// TIA Portal V14 SP1 export
// export: Created 2019-08-12T05:39:51.1994735Z, ExportSetting WithDefaults, WithReadOnly, DisplayName Totally Integrated Automation Portal, DisplayVersion V14 SP1 Update 6, DisplayName TIA Portal Openness, DisplayVersion V14 SP1 Update 6, DisplayName STEP 7 Professional, DisplayVersion V14 SP1 Update 6, DisplayName WinCC Professional, DisplayVersion V14 SP1 Update 6
FUNCTION_BLOCK "181M_Vibrating_screen"   // FB2008, LAD
TITLE = Управление виброситом силосов муки
{ S7_Optimized_Access := 'FALSE' }
VERSION : 0.1
// stored: AutoNumber false, CodeModifiedDate 2019-08-12T05:39:33.4572424Z, CompileDate 2019-08-12T05:39:33.4572423Z, CreationDate 2019-02-26T05:18:41.6523018Z, InterfaceModifiedDate 2019-08-09T12:59:29.73599Z, IsConsistent true, IsIECCheckEnabled false, IsKnowHowProtected false, ISMultiInstanceCapable true, IsWriteProtected false, LibraryConformanceStatus Warning: The object contains access to global data blocks. Warning: The block contains direct access to inputs, outputs, bit memories, indirect access to the registry or indirect access to external memory areas that are unknown at the time of compilation., ModifiedDate 2019-08-12T05:39:33.4572424Z, ParameterModified 2018-04-23T08:12:13.0838357Z, StructureModified 2019-08-09T12:59:29.73599Z, UDAEnableTagReadback false
   VAR DB_SPECIFIC
      HMI : Struct
         CMD : Struct
            Rot_FWD : Bool;   // Команда Вращение вперёд
            Stop : Bool;   // Команда Стоп
            Rot_BWD : Bool;   // Команда Вращение назад
            Spare_3 : Bool;
            Spare_4 : Bool;
            Spare_5 : Bool;
            Manual : Bool;   // Ручной режим
            Reset_Error : Bool;   // Сброс ошибок
         END_STRUCT;
         DATA : Struct
            StatusWord : Word;
            ContFbk1_Time : DInt := 4;   // Время контроля срабатывания контактора 1 / Время контроля срабатывания контактора 1 (сек)
            ContFbk2_Time : DInt := 4;   // Время контроля срабатывания контактора 2 / Время контроля срабатывания контактора 2 (сек)
            Rot_Off_Time : Int;   // Обратный отсчет времени остановки
            Warn_Not_Open_Valve : Bool;   // Сообщение о запуске очистки при закрытом клапане
            Warn_Not_Close_Valve : Bool;   // Сообщение о запуске работы при открытом клапане
         END_STRUCT;
      END_STRUCT;
   END_VAR
   VAR
      Two_Motor : "TwoMotorManag";
      TOF_Rot_FWD : TOF;
      TOF_Rot_REV : TOF;
   END_VAR
   VAR DB_SPECIFIC
      ContFbk1_Time : Time;   // Время контроля срабатывания контактора 1
      ContFbk2_Time : Time;   // Время контроля срабатывания контактора 2
      StopTime : Time;   // Время остановки мотора после вращения
      ResetErr : Bool;   // сброс ошибок
      General_cond_OK : Bool;   // Разрешение работы
      ManCmd_FWD : Bool;   // Команда ручного включения вращение вперёд
      ManCmd_REV : Bool;   // Команда ручного включения вращение назад
      ManCmd_Stop : Bool;   // Стоп
      AutoCmd_FWD : Bool;   // Команда автом. включения вращение вперёд
      AutoCmd_REV : Bool;   // Команда автом. включения вращение назад
      Spare : Bool;
      Spare_1 : Bool;
      Spare_2 : Bool;
      Spare_3 : Bool;
      Spare_4 : Bool;
      Spare_5 : Bool;
   END_VAR
   VAR_TEMP
      Temp_DINT : DInt;
   END_VAR
   VAR_TEMP   // added for the SCL form of the ladder/FBD networks
      _w1 : Bool;
   END_VAR
BEGIN

REGION Network 1: Сброс ошибок
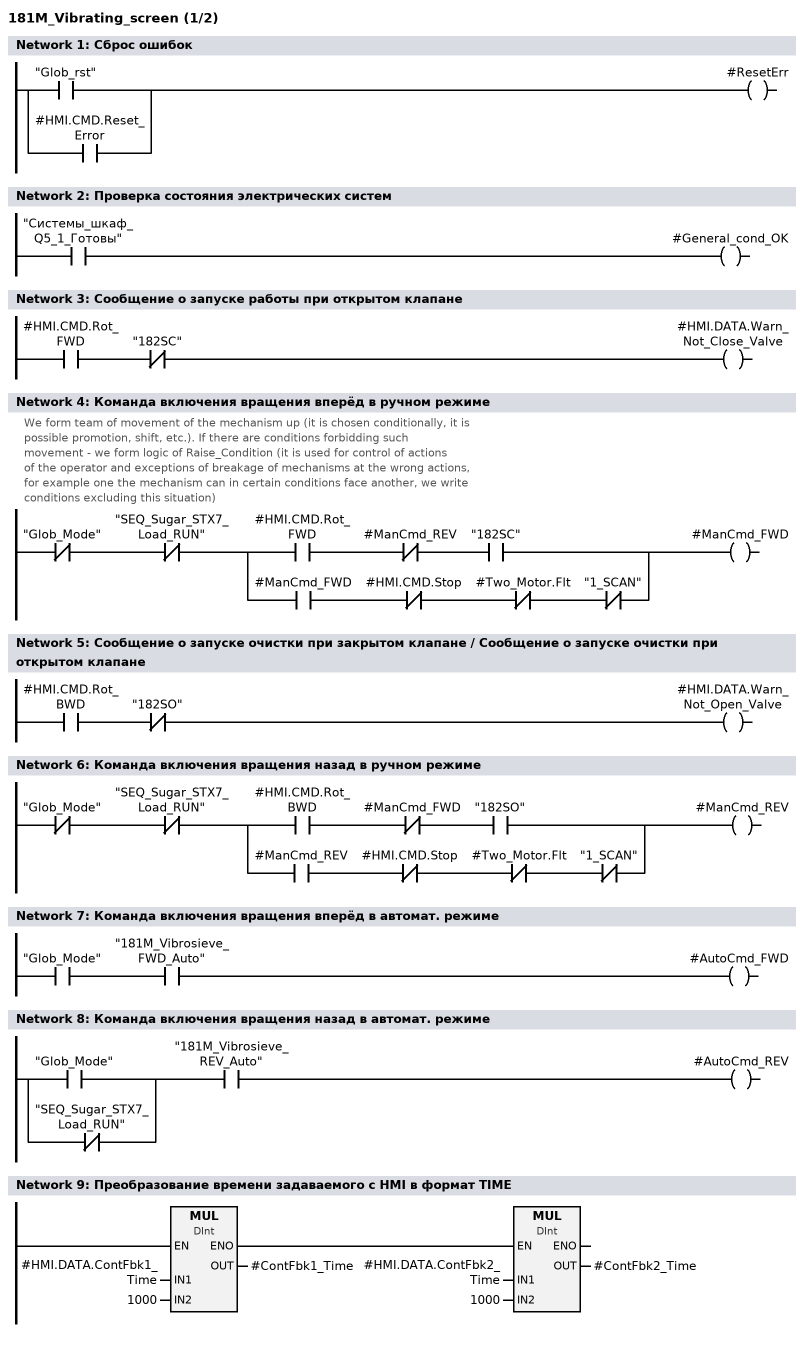
   RUNG wire#powerrail
      Contact( "Glob_rst" )
      wire#w1
      Coil( #ResetErr )
   END_RUNG
   RUNG wire#powerrail
      Contact( #HMI.CMD.Reset_Error )
   END_RUNG wire#w1
   // the same network as SCL:
   #ResetErr := "Glob_rst" OR #HMI.CMD.Reset_Error;
END_REGION

REGION Network 2: Проверка состояния электрических систем
   RUNG wire#powerrail
      Contact( "Системы_шкаф_Q5_1_Готовы" )
      Coil( #General_cond_OK )
   END_RUNG
   // the same network as SCL:
   #General_cond_OK := "Системы_шкаф_Q5_1_Готовы";
END_REGION

REGION Network 3: Сообщение о запуске работы при открытом клапане
   RUNG wire#powerrail
      Contact( #HMI.CMD.Rot_FWD )
      I_Contact( "182SC" )
      Coil( #HMI.DATA.Warn_Not_Close_Valve )
   END_RUNG
   // the same network as SCL:
   #HMI.DATA.Warn_Not_Close_Valve := #HMI.CMD.Rot_FWD AND NOT "182SC";
END_REGION

REGION Network 4: Команда включения вращения вперёд в ручном режиме
   // We form team of movement of the mechanism up (it is chosen conditionally, it is 
   // possible promotion, shift, etc.). If there are conditions forbidding such 
   // movement - we form logic of Raise_Condition (it is used for control of actions 
   // of the operator and exceptions of breakage of mechanisms at the wrong actions, 
   // for example one the mechanism can in certain conditions face another, we write 
   // conditions excluding this situation)
   RUNG wire#powerrail
      I_Contact( "Glob_Mode" )
      I_Contact( "SEQ_Sugar_STX7_Load_RUN" )
      wire#w1
      Contact( #HMI.CMD.Rot_FWD )
      I_Contact( #ManCmd_REV )
      Contact( "182SC" )
      wire#w2
      Coil( #ManCmd_FWD )
   END_RUNG
   RUNG wire#w1
      Contact( #ManCmd_FWD )
      I_Contact( #HMI.CMD.Stop )
      I_Contact( #Two_Motor.Flt )
      I_Contact( "1_SCAN" )
   END_RUNG wire#w2
   // the same network as SCL:
   #ManCmd_FWD := NOT "Glob_Mode" AND NOT "SEQ_Sugar_STX7_Load_RUN" AND ((#HMI.CMD.Rot_FWD AND NOT #ManCmd_REV AND "182SC") OR (#ManCmd_FWD AND NOT #HMI.CMD.Stop AND NOT #Two_Motor.Flt AND NOT "1_SCAN"));
END_REGION

REGION Network 5: Сообщение о запуске очистки при закрытом клапане / Сообщение о запуске очистки при открытом клапане
   RUNG wire#powerrail
      Contact( #HMI.CMD.Rot_BWD )
      I_Contact( "182SO" )
      Coil( #HMI.DATA.Warn_Not_Open_Valve )
   END_RUNG
   // the same network as SCL:
   #HMI.DATA.Warn_Not_Open_Valve := #HMI.CMD.Rot_BWD AND NOT "182SO";
END_REGION

REGION Network 6: Команда включения вращения назад в ручном режиме
   RUNG wire#powerrail
      I_Contact( "Glob_Mode" )
      I_Contact( "SEQ_Sugar_STX7_Load_RUN" )
      wire#w1
      Contact( #HMI.CMD.Rot_BWD )
      I_Contact( #ManCmd_FWD )
      Contact( "182SO" )
      wire#w2
      Coil( #ManCmd_REV )
   END_RUNG
   RUNG wire#w1
      Contact( #ManCmd_REV )
      I_Contact( #HMI.CMD.Stop )
      I_Contact( #Two_Motor.Flt )
      I_Contact( "1_SCAN" )
   END_RUNG wire#w2
   // the same network as SCL:
   #ManCmd_REV := NOT "Glob_Mode" AND NOT "SEQ_Sugar_STX7_Load_RUN" AND ((#HMI.CMD.Rot_BWD AND NOT #ManCmd_FWD AND "182SO") OR (#ManCmd_REV AND NOT #HMI.CMD.Stop AND NOT #Two_Motor.Flt AND NOT "1_SCAN"));
END_REGION

REGION Network 7: Команда включения вращения вперёд в автомат. режиме
   RUNG wire#powerrail
      Contact( "Glob_Mode" )
      Contact( "181M_Vibrosieve_FWD_Auto" )
      Coil( #AutoCmd_FWD )
   END_RUNG
   // the same network as SCL:
   #AutoCmd_FWD := "Glob_Mode" AND "181M_Vibrosieve_FWD_Auto";
END_REGION

REGION Network 8: Команда включения вращения назад в автомат. режиме
   RUNG wire#powerrail
      Contact( "Glob_Mode" )
      wire#w1
      Contact( "181M_Vibrosieve_REV_Auto" )
      Coil( #AutoCmd_REV )
   END_RUNG
   RUNG wire#powerrail
      I_Contact( "SEQ_Sugar_STX7_Load_RUN" )
   END_RUNG wire#w1
   // the same network as SCL:
   #AutoCmd_REV := ("Glob_Mode" OR NOT "SEQ_Sugar_STX7_Load_RUN") AND "181M_Vibrosieve_REV_Auto";
END_REGION

REGION Network 9: Преобразование времени задаваемого с HMI в формат TIME
   RUNG wire#powerrail
      { S7_Templates := "SrcType := DInt"; S7_GenerateENO := "TRUE" } Mul(in1 := #HMI.DATA.ContFbk1_Time, in2 := 1000, out => #ContFbk1_Time)
      { S7_Templates := "SrcType := DInt"; S7_GenerateENO := "TRUE" } Mul(in1 := #HMI.DATA.ContFbk2_Time, in2 := 1000, out => #ContFbk2_Time)
   END_RUNG
   // the same network as SCL:
   // ENO of a box is taken as its EN; it also drops when the box reports an error
   #ContFbk1_Time := #HMI.DATA.ContFbk1_Time * 1000;
   #ContFbk2_Time := #HMI.DATA.ContFbk2_Time * 1000;
END_REGION

REGION Network 10: Время остановки мотора
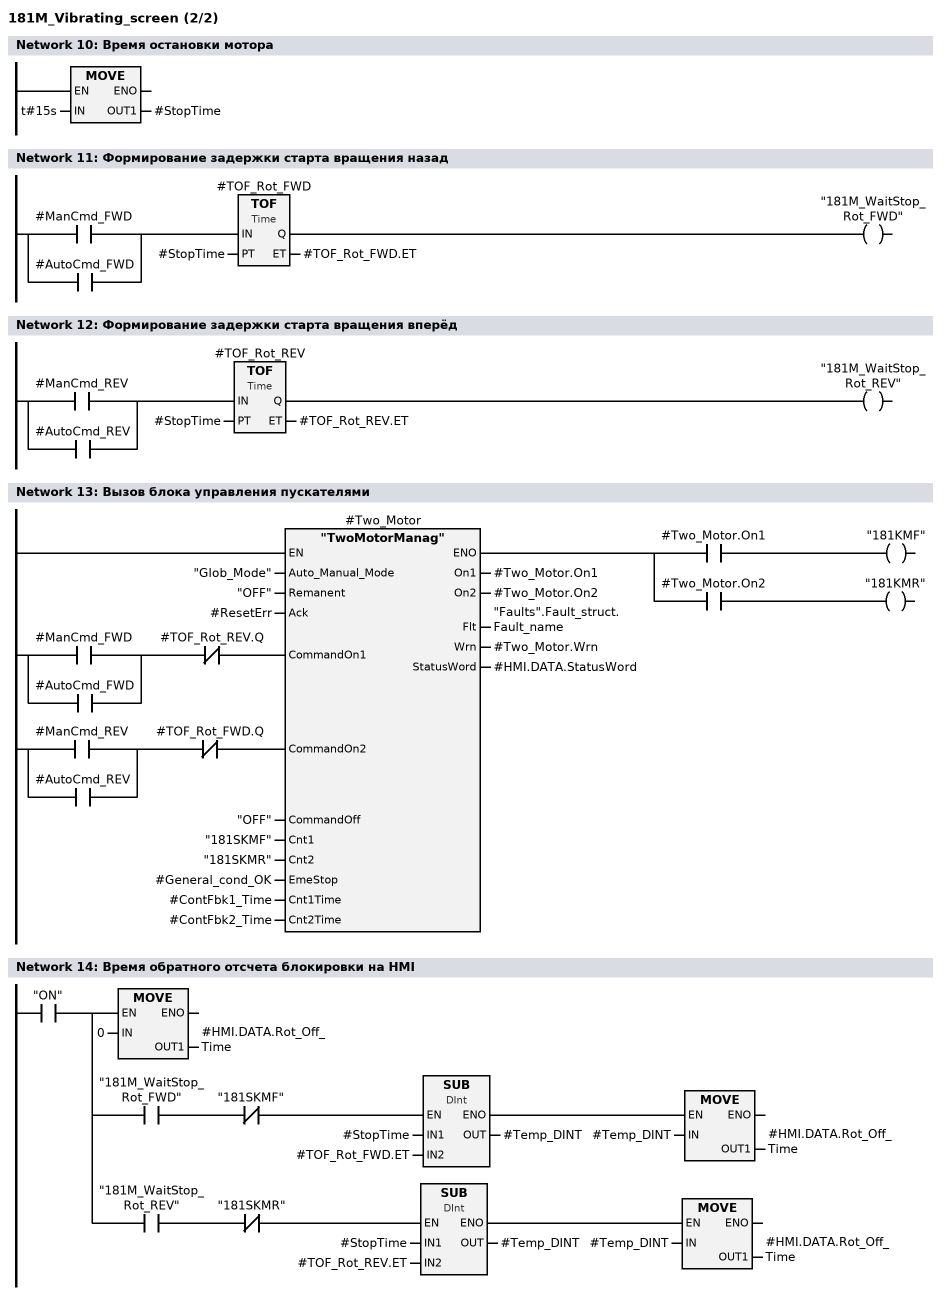
   RUNG wire#powerrail
      { S7_GenerateENO := "TRUE" } Move(in := t#15s, out1 => #StopTime)
   END_RUNG
   // the same network as SCL:
   #StopTime := t#15s;
END_REGION

REGION Network 11: Формирование задержки старта вращения назад
   RUNG wire#powerrail
      Contact( #ManCmd_FWD )
      wire#w1
      { S7_Templates := "time_type := Time" } #TOF_Rot_FWD.TOF(pt := #StopTime, et => #TOF_Rot_FWD.ET)
      Coil( "181M_WaitStop_Rot_FWD" )
   END_RUNG
   RUNG wire#powerrail
      Contact( #AutoCmd_FWD )
   END_RUNG wire#w1
   // the same network as SCL:
   #TOF_Rot_FWD.TOF(IN := #ManCmd_FWD OR #AutoCmd_FWD, PT := #StopTime, ET => #TOF_Rot_FWD.ET);
   "181M_WaitStop_Rot_FWD" := #TOF_Rot_FWD.Q;
END_REGION

REGION Network 12: Формирование задержки старта вращения вперёд
   RUNG wire#powerrail
      Contact( #ManCmd_REV )
      wire#w1
      { S7_Templates := "time_type := Time" } #TOF_Rot_REV.TOF(pt := #StopTime, et => #TOF_Rot_REV.ET)
      Coil( "181M_WaitStop_Rot_REV" )
   END_RUNG
   RUNG wire#powerrail
      Contact( #AutoCmd_REV )
   END_RUNG wire#w1
   // the same network as SCL:
   #TOF_Rot_REV.TOF(IN := #ManCmd_REV OR #AutoCmd_REV, PT := #StopTime, ET => #TOF_Rot_REV.ET);
   "181M_WaitStop_Rot_REV" := #TOF_Rot_REV.Q;
END_REGION

REGION Network 13: Вызов блока управления пускателями
   RUNG wire#powerrail
      #Two_Motor(CommandOn1 := wire#w2, CommandOn2 := wire#w4, Auto_Manual_Mode := "Glob_Mode", Remanent := "OFF", Ack := #ResetErr, CommandOff := "OFF", Cnt1 := "181SKMF", Cnt2 := "181SKMR", EmeStop := #General_cond_OK, Cnt1Time := #ContFbk1_Time, Cnt2Time := #ContFbk2_Time, On1 => #Two_Motor.On1, On2 => #Two_Motor.On2, Flt => "Faults".Fault_struct.Fault_name, Wrn => #Two_Motor.Wrn, StatusWord => #HMI.DATA.StatusWord)
      wire#w5
      Contact( #Two_Motor.On1 )
      Coil( "181KMF" )
   END_RUNG
   RUNG wire#powerrail
      Contact( #ManCmd_FWD )
      wire#w1
      I_Contact( #TOF_Rot_REV.Q )
   END_RUNG wire#w2
   RUNG wire#powerrail
      Contact( #AutoCmd_FWD )
   END_RUNG wire#w1
   RUNG wire#powerrail
      Contact( #ManCmd_REV )
      wire#w3
      I_Contact( #TOF_Rot_FWD.Q )
   END_RUNG wire#w4
   RUNG wire#powerrail
      Contact( #AutoCmd_REV )
   END_RUNG wire#w3
   RUNG wire#w5
      Contact( #Two_Motor.On2 )
      Coil( "181KMR" )
   END_RUNG
   // the same network as SCL:
   #Two_Motor(Auto_Manual_Mode := "Glob_Mode",   // "TwoMotorManag"
              Remanent := "OFF",
              Ack := #ResetErr,
              CommandOn1 := (#ManCmd_FWD OR #AutoCmd_FWD) AND NOT #TOF_Rot_REV.Q,
              CommandOn2 := (#ManCmd_REV OR #AutoCmd_REV) AND NOT #TOF_Rot_FWD.Q,
              CommandOff := "OFF",
              Cnt1 := "181SKMF",
              Cnt2 := "181SKMR",
              EmeStop := #General_cond_OK,
              Cnt1Time := #ContFbk1_Time,
              Cnt2Time := #ContFbk2_Time,
              On1 => #Two_Motor.On1,
              On2 => #Two_Motor.On2,
              Flt => "Faults".Fault_struct.Fault_name,
              Wrn => #Two_Motor.Wrn,
              StatusWord => #HMI.DATA.StatusWord,
              ENO => #_w1);
   "181KMF" := #_w1 AND #Two_Motor.On1;
   "181KMR" := #_w1 AND #Two_Motor.On2;
END_REGION

REGION Network 14: Время обратного отсчета блокировки на HMI
   RUNG wire#powerrail
      Contact( "ON" )
      wire#w1
      { S7_GenerateENO := "TRUE" } Move(in := 0, out1 => #HMI.DATA.Rot_Off_Time)
   END_RUNG
   RUNG wire#w1
      Contact( "181M_WaitStop_Rot_FWD" )
      I_Contact( "181SKMF" )
      { S7_Templates := "SrcType := DInt"; S7_GenerateENO := "TRUE" } Sub(in1 := #StopTime, in2 := #TOF_Rot_FWD.ET, out => #Temp_DINT)
      { S7_GenerateENO := "TRUE" } Move(in := #Temp_DINT, out1 => #HMI.DATA.Rot_Off_Time)
   END_RUNG
   RUNG wire#w1
      Contact( "181M_WaitStop_Rot_REV" )
      I_Contact( "181SKMR" )
      { S7_Templates := "SrcType := DInt"; S7_GenerateENO := "TRUE" } Sub(in1 := #StopTime, in2 := #TOF_Rot_REV.ET, out => #Temp_DINT)
      { S7_GenerateENO := "TRUE" } Move(in := #Temp_DINT, out1 => #HMI.DATA.Rot_Off_Time)
   END_RUNG
   // the same network as SCL:
   // ENO of a box is taken as its EN; it also drops when the box reports an error
   IF "ON" THEN #HMI.DATA.Rot_Off_Time := 0; END_IF;
   IF "ON" AND "181M_WaitStop_Rot_FWD" AND NOT "181SKMF" THEN
       #Temp_DINT := #StopTime - #TOF_Rot_FWD.ET;
       #HMI.DATA.Rot_Off_Time := #Temp_DINT;
   END_IF;
   IF "ON" AND "181M_WaitStop_Rot_REV" AND NOT "181SKMR" THEN
       #Temp_DINT := #StopTime - #TOF_Rot_REV.ET;
       #HMI.DATA.Rot_Off_Time := #Temp_DINT;
   END_IF;
END_REGION
END_FUNCTION_BLOCK
